FUNCTION TO_LSTRING : LSTRING
VAR_INPUT
  str: STRING(255);
END_VAR
VAR
END_VAR

TO_LSTRING.str := str;

END_FUNCTION

(* stored: Version 1.1.0.1, ProductVersion 3.1.4024.9
   POU TO_LSTRING: Id {f368814f-f5b3-4c61-998a-cd6abeb4f954}, SpecialFunc None *)
